PROGRAM MAIN
VAR
	
END_VAR

PI_CNTRL_SIM_CLOSED_LOOP();

END_PROGRAM

(* stored: Version 1.1.0.1, ProductVersion 3.1.4024.9
   POU MAIN: Id {d3da440d-be59-4f15-8a72-cab117e406ce}, SpecialFunc None *)
